INTERFACE IExecution

METHOD Abort 
VAR_INPUT
END_VAR
END_METHOD

PROPERTY Aborted : BOOL
GET
END_GET
END_PROPERTY

PROPERTY Busy : BOOL
GET
END_GET
END_PROPERTY

METHOD Clear 
VAR_INPUT
END_VAR
END_METHOD

PROPERTY Done : BOOL
GET
END_GET
END_PROPERTY

PROPERTY Error : BOOL
GET
END_GET
END_PROPERTY

PROPERTY ErrorId : UDINT
GET
END_GET
END_PROPERTY

PROPERTY Event_OnAbort : IEvent
GET
END_GET
SET
END_SET
END_PROPERTY

PROPERTY Event_OnError : IEvent
GET
END_GET
SET
END_SET
END_PROPERTY

PROPERTY Ready : BOOL
GET
END_GET
END_PROPERTY

METHOD Start : BOOL // returns TRUE if start request accepted (i.e State was Ready)
VAR_INPUT
END_VAR
END_METHOD

PROPERTY Starting : BOOL
GET
END_GET
END_PROPERTY

END_INTERFACE

(* stored: Version 1.1.0.1, ProductVersion 3.1.4024.3
   Itf IExecution: Id {2e2a9e90-2894-0caa-065e-86441183945f}
   Folder Methods: Id {4df2c49f-ecc5-41ac-a5f7-eb029ec847e7}
   Folder Properties: Id {858ea4b7-fbd7-4d4c-a650-4ab711825959}
   Method Abort: Id {b913466c-26cf-0433-3b1e-51d91dedf168}
   Property Aborted: Id {5347566a-e4a6-4028-bbdd-c7c385fe1cab}
   Get Get: Id {68b612a5-196e-4381-a504-106ddf11c80e}
   Property Busy: Id {6cebbaf7-86c1-4b42-b741-1563ee9a82a3}
   Get Get: Id {c2417d08-69f5-4b45-8674-471ac6e75ca8}
   Method Clear: Id {58de2a78-426c-4017-a46d-fddd798e420e}
   Property Done: Id {f19ffc53-eaf1-48be-aca7-f281232899dc}
   Get Get: Id {06415348-1825-402b-9b90-995ba15a6503}
   Property Error: Id {54cfaecc-395a-4685-8d6b-701b343961c9}
   Get Get: Id {cff8eb45-644a-457e-91bd-f88883679daa}
   Property ErrorId: Id {554c0d62-de61-4cee-b138-02830007f416}
   Get Get: Id {3988269b-c4af-4b43-b25b-132866f150af}
   Property Event_OnAbort: Id {aa6718e5-a154-4d63-b597-d56558a437a2}
   Get Get: Id {9b4d3ced-e6a5-451e-a1ce-71ba48bbfe04}
   Set Set: Id {4588cfbb-42b1-4cab-b5f2-67f8502177ce}
   Property Event_OnError: Id {f7d42420-ef1e-476e-96d6-701a9a01a5ba}
   Get Get: Id {83bf764f-a383-412c-8d91-57d70eec55af}
   Set Set: Id {d2c49168-cc52-44a9-bce6-660c347d836d}
   Property Ready: Id {b91ada47-a851-4255-ace3-07ff2a4d3deb}
   Get Get: Id {bde8a44c-e6cd-483a-a94e-c0d4f73a98b1}
   Method Start: Id {28e25cff-ad88-0708-05e8-5a4e484e10dc}
   Property Starting: Id {6b02f8f3-9828-4ea0-8253-65483424421e}
   Get Get: Id {d6faa71d-a2a3-4abf-8c36-46cccd4f90e4} *)
